// Provide logging 
FUNCTION_BLOCK FB_FileLogging IMPLEMENTS I_Logging
VAR_INPUT
	eLogLevel:				E_LogLevel:= E_LogLevel.Verbose;
END_VAR
VAR_OUTPUT
END_VAR
VAR
	iLogging:				I_Logging;
END_VAR

METHOD PUBLIC M_Attach : BOOL
VAR_INPUT
	iLogging:				I_Logging;
END_VAR
IF THIS^.iLogging = 0 THEN
	THIS^.iLogging:= iLogging;
	M_Attach:= TRUE;
ELSIF THIS^.iLogging = iLogging THEN
	// already inside
	M_Attach:= TRUE;
	RETURN;
ELSE
	// redirect to next logging function block
	THIS^.iLogging.M_Attach(iLogging);
END_IF
END_METHOD

METHOD PUBLIC M_Log : BOOL
VAR_INPUT
	eLogLevel:			E_LogLevel;
	nID:				UDINT;
	sSource:			STRING(255);
	sMessage:			STRING(255);
	sArguments:			STRING(255);
END_VAR
VAR
	fbMsg:				FB_TcLogging; 
	fbSourceInfo:		FB_TcSourceInfo;
END_VAR
END_METHOD

PROPERTY PUBLIC P_LogLevel : E_LogLevel
GET
P_LogLevel:= eLogLevel;
END_GET
SET
eLogLevel:= P_LogLevel;
END_SET
END_PROPERTY

END_FUNCTION_BLOCK

(* stored: Version 1.1.0.1
   POU FB_FileLogging: Id {98718708-3849-429d-beae-f0d90c92980c}, SpecialFunc None
   Method M_Attach: Id {e5f3d61e-3e1e-49a5-be36-d112b991237f}
   Method M_Log: Id {99ec6938-a1ad-4754-8b3a-271a0cd755f4}
   Property P_LogLevel: Id {e44967b0-7bc6-4691-a053-a7a9ae307d31}
   Get Get: Id {a7b9af1e-350a-4368-9af9-ad37be55cf9f}
   Set Set: Id {ee7c41e7-11fd-4dce-aade-31ad3f7ed8fc} *)
